{attribute 'linkalways'} 
{attribute 'no_explicit_call' := 'This FB is a CLASS and must be accessed using methods or properties'}
{attribute 'enable_dynamic_creation'}
FUNCTION_BLOCK Node_F_VN_BitwiseOrVectorWithImage EXTENDS VisionNode
VAR
    aVector : _TcVnVector4_LREAL;
    ipSrcImage : _ITcVnImage;
    ipDestImage : _ITcVnImage;
    hrPrev : _HRESULT(S_OK);
	hresult : _HRESULT(S_OK);
END_VAR

METHOD PUBLIC  Clone : I_Node
VAR
	pNode : POINTER TO Node_F_VN_BitwiseOrVectorWithImage;
END_VAR
pNode := __NEW(Node_F_VN_BitwiseOrVectorWithImage);
Clone := pNode^;
END_METHOD

METHOD FB_init : BOOL
VAR_INPUT
	bInitRetains : BOOL; // if TRUE, the retain variables are initialized (warm start / cold start)
	bInCopyCode : BOOL;  // if TRUE, the instance afterwards gets moved into the copy code (online change)
END_VAR
AddInput('aVector', aVector);
AddInput('ipSrcImage', ipSrcImage);
AddInput('hrPrev', hrPrev);
AddOutput('ipDestImage', ipDestImage);
AddOutput('hresult',hresult);
END_METHOD

METHOD PROTECTED OnExecute : HRESULT
hresult.Value := F_VN_BitwiseOrVectorWithImage(
    aVector := aVector.Value,
    ipSrcImage := ipSrcImage.Value,
	ipDestImage := ipDestImage.Value,
	hrPrev:= hrPrev.Value);
END_METHOD

METHOD PUBLIC PreExecutionCheck
VAR_INPUT
	Check : I_PreExecutionChecks;
END_VAR
Check.IsTrue(ipSrcImage.IsValid, 'ipSrcImage must contain an image');
END_METHOD

END_FUNCTION_BLOCK

(* stored: Version 1.1.0.1, ProductVersion 3.1.4024.13
   POU Node_F_VN_BitwiseOrVectorWithImage: Id {b1c7d500-cb7e-0305-3ed8-af3ce6dd8bfa}, SpecialFunc None
   Folder Constructor: Id {2738ad2a-e1f5-01f1-3e65-3f6e6fa0eea4}
   Method Clone: Id {5a2e6a38-fcbf-0878-016e-cb5afd227825}
   Method FB_init: Id {0d55c965-af21-0f85-05d5-88ca49e8084a}
   Method OnExecute: Id {cc04444b-5473-095f-070f-81722b7b113f}
   Method PreExecutionCheck: Id {a8aaf6d2-7837-01f7-10d2-c8dc564c3870} *)
